Staubli VAL3: cycle_getProg.pgx

program cycle_getProg(string& x_sName[] (dimensions=1), num x_nIndex (dimensions=1), num x_nType (dimensions=1))
  local num l_nID
  local num l_nSize[3]
begin
  //
  // get the programm name of the specific
  // x_nIndex, return "" if there is an error
  // x_nIndex start from 1 o N
  //
  if saveData:bDebug
    ? "[KERNEL] PLC:Ask program name at index:"+toString("",x_nIndex)
  endIf
  call cycle_getSize(l_nSize,x_nType)
  if x_nIndex<=l_nSize and x_nIndex>0
    l_nID=0
    call processList:getCycle(x_sName,l_nID,l_nID,x_nIndex-1,x_nType)
  else
    logMsg("[KERNEL] PLC: "+x_sName+" error on the index "+toString("",x_nIndex))
    x_sName=""
  endIf
end
